FUNCTION_BLOCK EL3122
VAR
	_io : EL3xx2_Data;
	{attribute addProperty Name "WcState"}
	_wcState : WcStateInputToggle;
	{attribute addProperty Name "Info data"}
	_infoData : InfoDataAds;
END_VAR

PROPERTY IO : REFERENCE TO EL3xx2_Data
GET
IO REF= _io;
END_GET
END_PROPERTY

PROPERTY WcState : REFERENCE TO WcStateInputToggle
GET
WcState REF= _wcState;
END_GET
END_PROPERTY

END_FUNCTION_BLOCK

(* stored: Version 1.1.0.1, ProductVersion 3.1.4024.9
   POU EL3122: Id {bbd90905-0357-0dd3-36ac-4314bf1e11dc}, SpecialFunc None
   Property IO: Id {74426593-7879-0fe3-04ed-2cee96338342}
   Get Get: Id {8809362f-a07c-0aa5-0981-977a3ff6fb7a}
   Property WcState: Id {f011d0ea-6c68-0877-079e-0113602a4743}
   Get Get: Id {f7972d1c-9f1c-0a90-0d5e-9ff21cc71a71} *)
